TYPE ST_Sensors :
STRUCT
END_STRUCT
END_TYPE

(* stored: Version 1.1.0.1, ProductVersion 3.1.4024.12
   DUT ST_Sensors: Id {f7cf5bf2-baaf-4f6d-8ec9-9aee307292ac} *)
